FUNCTION_BLOCK RIDGE_MODEL
  {SET_ATTRIBUTE(OpcUa, SERVICE)}
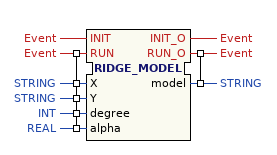
  EVENT_INPUT
    INIT;
    RUN WITH X, Y, degree, alpha; {SET_ATTRIBUTE(OpcUa, Method)}
  END_EVENT
  EVENT_OUTPUT
    INIT_O;
    RUN_O WITH model;
  END_EVENT
  VAR_INPUT
    X : STRING; {SET_ATTRIBUTE(OpcUa, Variable.RUN)}
    Y : STRING; {SET_ATTRIBUTE(OpcUa, Variable.RUN)}
    degree : INT; {SET_ATTRIBUTE(OpcUa, Variable.RUN)}
    alpha : REAL; {SET_ATTRIBUTE(OpcUa, Variable.RUN)}
  END_VAR
  VAR_OUTPUT
    model : STRING; {SET_ATTRIBUTE(OpcUa, Variable.RUN)}
  END_VAR
END_FUNCTION_BLOCK
